INTERFACE I_Vector EXTENDS I_Object

METHOD ToArray : ARRAY[0..2] OF LREAL
VAR_INPUT
END_VAR
END_METHOD

PROPERTY X : LREAL
GET
END_GET
SET
END_SET
END_PROPERTY

PROPERTY Y : LREAL
GET
END_GET
SET
END_SET
END_PROPERTY

PROPERTY Z : LREAL
GET
END_GET
SET
END_SET
END_PROPERTY

END_INTERFACE

(* stored: Version 1.1.0.1, ProductVersion 3.1.4024.4
   Itf I_Vector: Id {a5b20593-58ec-488d-9d6c-09788d737ec4}
   Method ToArray: Id {c70895f5-952c-48db-b4f2-aeede81127d3}
   Property X: Id {98948d46-6fc2-4df3-9cc0-d075dedef1ef}
   Get Get: Id {ecc948c3-67ca-4aa1-a73c-91260d10a5f2}
   Set Set: Id {f3aab3e8-6fc2-4dfa-a706-f409d00872c0}
   Property Y: Id {a7d4c1d6-5eb9-4de6-98ac-2648803ecb8f}
   Get Get: Id {bb79637b-d797-4ff2-8461-b7e8190be576}
   Set Set: Id {7a237524-3af9-4d69-b66e-4aa0e8dc7c88}
   Property Z: Id {a25933c9-7092-4059-8208-e4c757079866}
   Get Get: Id {f289ea35-4814-493a-b466-831d89f66c22}
   Set Set: Id {fbe292cd-c146-4498-af9e-b4559e8f8e42} *)
